FUNCTION_BLOCK FB_LoadCell EXTENDS FB_SolidSamplingModule
VAR_INPUT
END_VAR
VAR_OUTPUT
END_VAR
VAR
END_VAR

END_FUNCTION_BLOCK

(* stored: Version 1.1.0.1
   POU FB_LoadCell: Id {4dc582d4-e063-44b6-9e44-474d705e88f5}, SpecialFunc None *)
